{attribute 'GeneratedUsingTerminal: EP2038-0001-0016'}
{attribute addProperty BoxType "EP2038-0001-0016"}
{attribute addProperty Id "InputAT %I*BOOL1"}
{attribute addProperty CRC "2198356929"}
{attribute addProperty Size "1"}
TYPE Diag_Channel_830843C1 EXTENDS InputBase_8311D824 :
STRUCT
	{attribute addProperty Name "Input"}
	Input AT %I* : BOOL;
END_STRUCT
END_TYPE

(* stored: Version 1.2.0.0, ProductVersion 3.1.4024.9
   DUT Diag_Channel_830843C1: Id {80063fa1-7dc1-4580-a610-8a926be0c258} *)
